{attribute 'qualified_only'}
VAR_GLOBAL
	bEndStopOverride : BOOL; 
END_VAR

(* stored: Version 1.1.0.1, ProductVersion 3.1.4026.11
   GVL HMI: Id {26f8b220-c366-427c-968e-e98e5cf6b52c} *)
